{attribute 'OPC.UA.DA.StructuredType' := '1'}
TYPE stBelt :
STRUCT
	sName		: STRING[10];
	uliOrder	: ULINT;
	xFull		: BOOL;
	xEmpty		: BOOL;
	xAvailable	: BOOL;
	xEnable		: BOOL;
END_STRUCT
END_TYPE

(* stored: Version 1.1.0.1, ProductVersion 3.1.4024.11
   DUT stBelt: Id {7d7f1f52-f09c-49e8-b6e4-c0880289f9f7} *)
